(* Logix 5000 project; controller DC01 vendor 1 type 14 code 165 rev 32.12; software revision 32.04; part 8 of 13 *)
(* tags used below, declared in another part *)
   Break1_Length : DINT;
   Break2_Length : DINT;
   Lunch_Length : DINT;
   null : STRING;
   LN03_Schedule : UDT_Current_Status;
   LN03_Weekly_Schedule : UDT_Weekly_Schedule;
(* LN03, continued *)

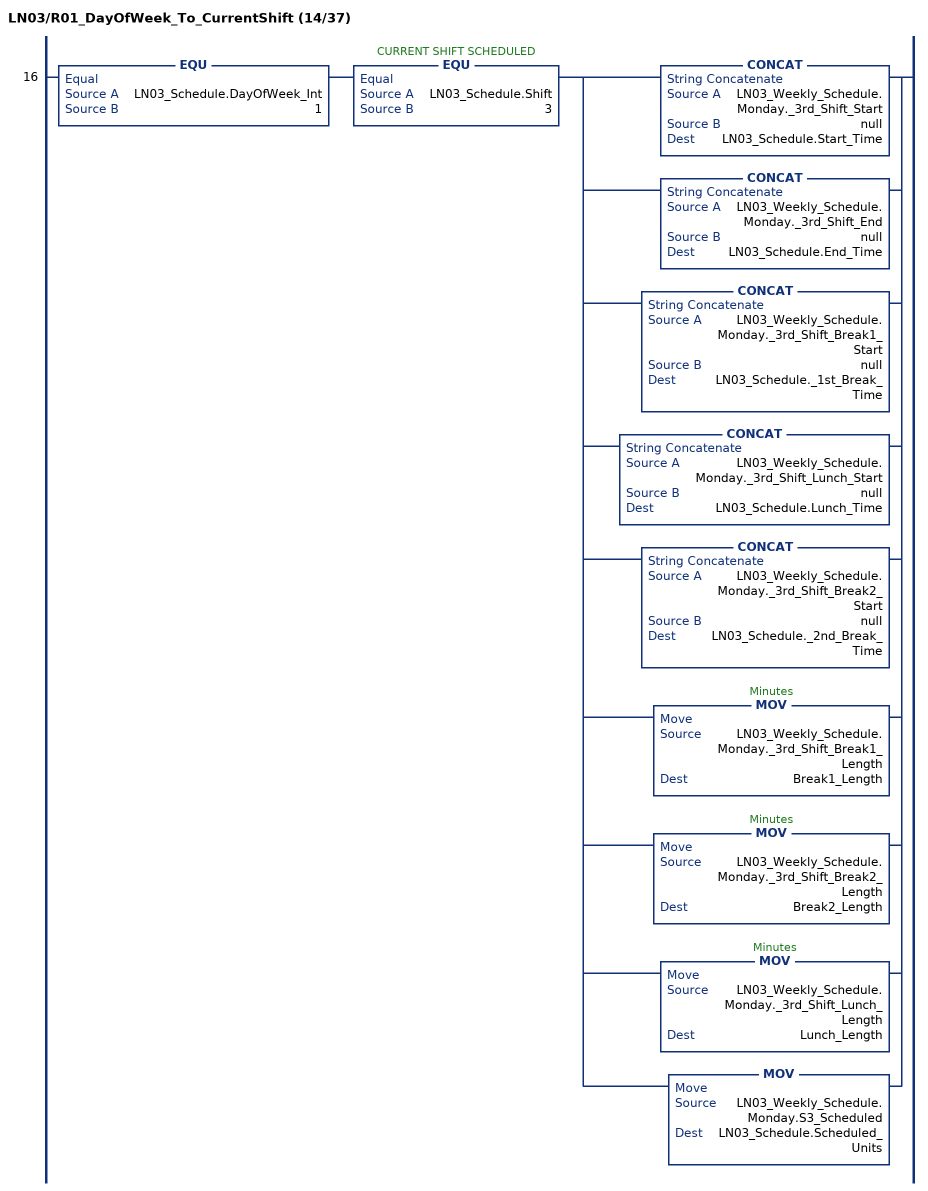
   [picture p147: LN03/R01_DayOfWeek_To_CurrentShift rungs 16-16]
   16: EQU(LN03_Schedule.DayOfWeek_Int,1)EQU(LN03_Schedule.Shift,3)[CONCAT(LN03_Weekly_Schedule.Monday._3rd_Shift_Start,null,LN03_Schedule.Start_Time) ,CONCAT(LN03_Weekly_Schedule.Monday._3rd_Shift_End,null,LN03_Schedule.End_Time) ,CONCAT(LN03_Weekly_Schedule.Monday._3rd_Shift_Break1_Start,null,LN03_Schedule._1st_Break_Time) ,CONCAT(LN03_Weekly_Schedule.Monday._3rd_Shift_Lunch_Start,null,LN03_Schedule.Lunch_Time) ,CONCAT(LN03_Weekly_Schedule.Monday._3rd_Shift_Break2_Start,null,LN03_Schedule._2nd_Break_Time) ,MOV(LN03_Weekly_Schedule.Monday._3rd_Shift_Break1_Length,Break1_Length) ,MOV(LN03_Weekly_Schedule.Monday._3rd_Shift_Break2_Length,Break2_Length) ,MOV(LN03_Weekly_Schedule.Monday._3rd_Shift_Lunch_Length,Lunch_Length) ,MOV(LN03_Weekly_Schedule.Monday.S3_Scheduled,LN03_Schedule.Scheduled_Units) ];
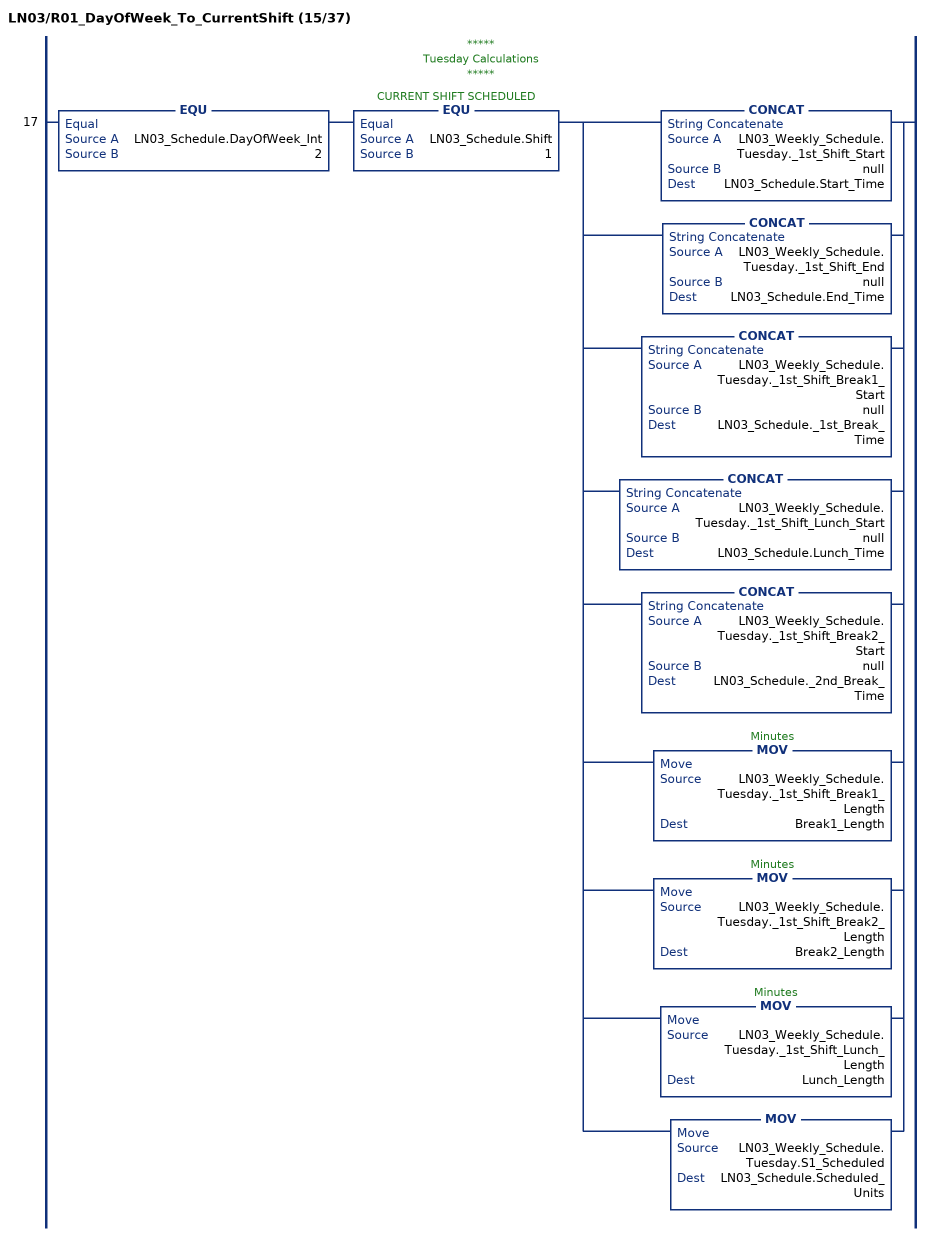
   // *****
   // Tuesday Calculations
   // *****
   17: EQU(LN03_Schedule.DayOfWeek_Int,2)EQU(LN03_Schedule.Shift,1)[CONCAT(LN03_Weekly_Schedule.Tuesday._1st_Shift_Start,null,LN03_Schedule.Start_Time) ,CONCAT(LN03_Weekly_Schedule.Tuesday._1st_Shift_End,null,LN03_Schedule.End_Time) ,CONCAT(LN03_Weekly_Schedule.Tuesday._1st_Shift_Break1_Start,null,LN03_Schedule._1st_Break_Time) ,CONCAT(LN03_Weekly_Schedule.Tuesday._1st_Shift_Lunch_Start,null,LN03_Schedule.Lunch_Time) ,CONCAT(LN03_Weekly_Schedule.Tuesday._1st_Shift_Break2_Start,null,LN03_Schedule._2nd_Break_Time) ,MOV(LN03_Weekly_Schedule.Tuesday._1st_Shift_Break1_Length,Break1_Length) ,MOV(LN03_Weekly_Schedule.Tuesday._1st_Shift_Break2_Length,Break2_Length) ,MOV(LN03_Weekly_Schedule.Tuesday._1st_Shift_Lunch_Length,Lunch_Length) ,MOV(LN03_Weekly_Schedule.Tuesday.S1_Scheduled,LN03_Schedule.Scheduled_Units) ];
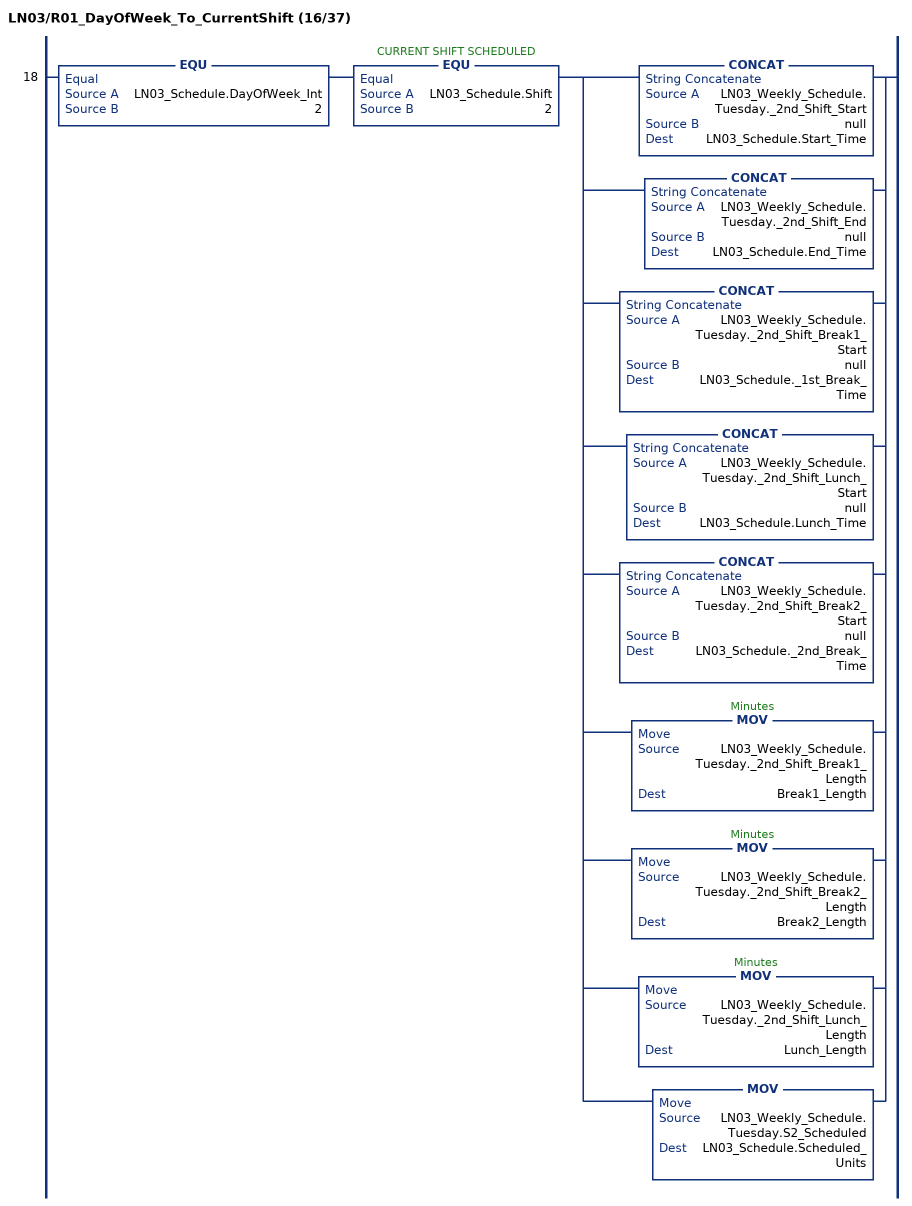
   18: EQU(LN03_Schedule.DayOfWeek_Int,2)EQU(LN03_Schedule.Shift,2)[CONCAT(LN03_Weekly_Schedule.Tuesday._2nd_Shift_Start,null,LN03_Schedule.Start_Time) ,CONCAT(LN03_Weekly_Schedule.Tuesday._2nd_Shift_End,null,LN03_Schedule.End_Time) ,CONCAT(LN03_Weekly_Schedule.Tuesday._2nd_Shift_Break1_Start,null,LN03_Schedule._1st_Break_Time) ,CONCAT(LN03_Weekly_Schedule.Tuesday._2nd_Shift_Lunch_Start,null,LN03_Schedule.Lunch_Time) ,CONCAT(LN03_Weekly_Schedule.Tuesday._2nd_Shift_Break2_Start,null,LN03_Schedule._2nd_Break_Time) ,MOV(LN03_Weekly_Schedule.Tuesday._2nd_Shift_Break1_Length,Break1_Length) ,MOV(LN03_Weekly_Schedule.Tuesday._2nd_Shift_Break2_Length,Break2_Length) ,MOV(LN03_Weekly_Schedule.Tuesday._2nd_Shift_Lunch_Length,Lunch_Length) ,MOV(LN03_Weekly_Schedule.Tuesday.S2_Scheduled,LN03_Schedule.Scheduled_Units) ];
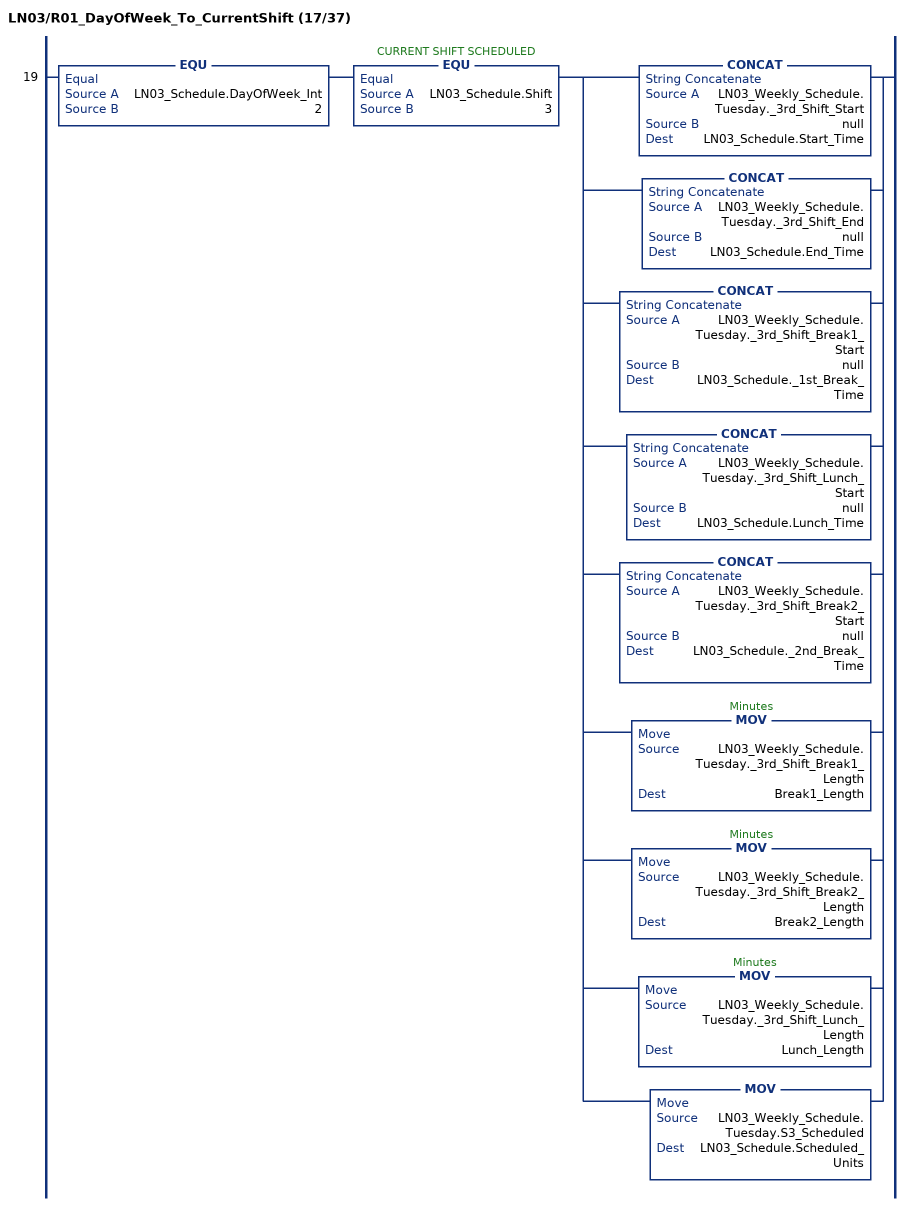
   19: EQU(LN03_Schedule.DayOfWeek_Int,2)EQU(LN03_Schedule.Shift,3)[CONCAT(LN03_Weekly_Schedule.Tuesday._3rd_Shift_Start,null,LN03_Schedule.Start_Time) ,CONCAT(LN03_Weekly_Schedule.Tuesday._3rd_Shift_End,null,LN03_Schedule.End_Time) ,CONCAT(LN03_Weekly_Schedule.Tuesday._3rd_Shift_Break1_Start,null,LN03_Schedule._1st_Break_Time) ,CONCAT(LN03_Weekly_Schedule.Tuesday._3rd_Shift_Lunch_Start,null,LN03_Schedule.Lunch_Time) ,CONCAT(LN03_Weekly_Schedule.Tuesday._3rd_Shift_Break2_Start,null,LN03_Schedule._2nd_Break_Time) ,MOV(LN03_Weekly_Schedule.Tuesday._3rd_Shift_Break1_Length,Break1_Length) ,MOV(LN03_Weekly_Schedule.Tuesday._3rd_Shift_Break2_Length,Break2_Length) ,MOV(LN03_Weekly_Schedule.Tuesday._3rd_Shift_Lunch_Length,Lunch_Length) ,MOV(LN03_Weekly_Schedule.Tuesday.S3_Scheduled,LN03_Schedule.Scheduled_Units) ];
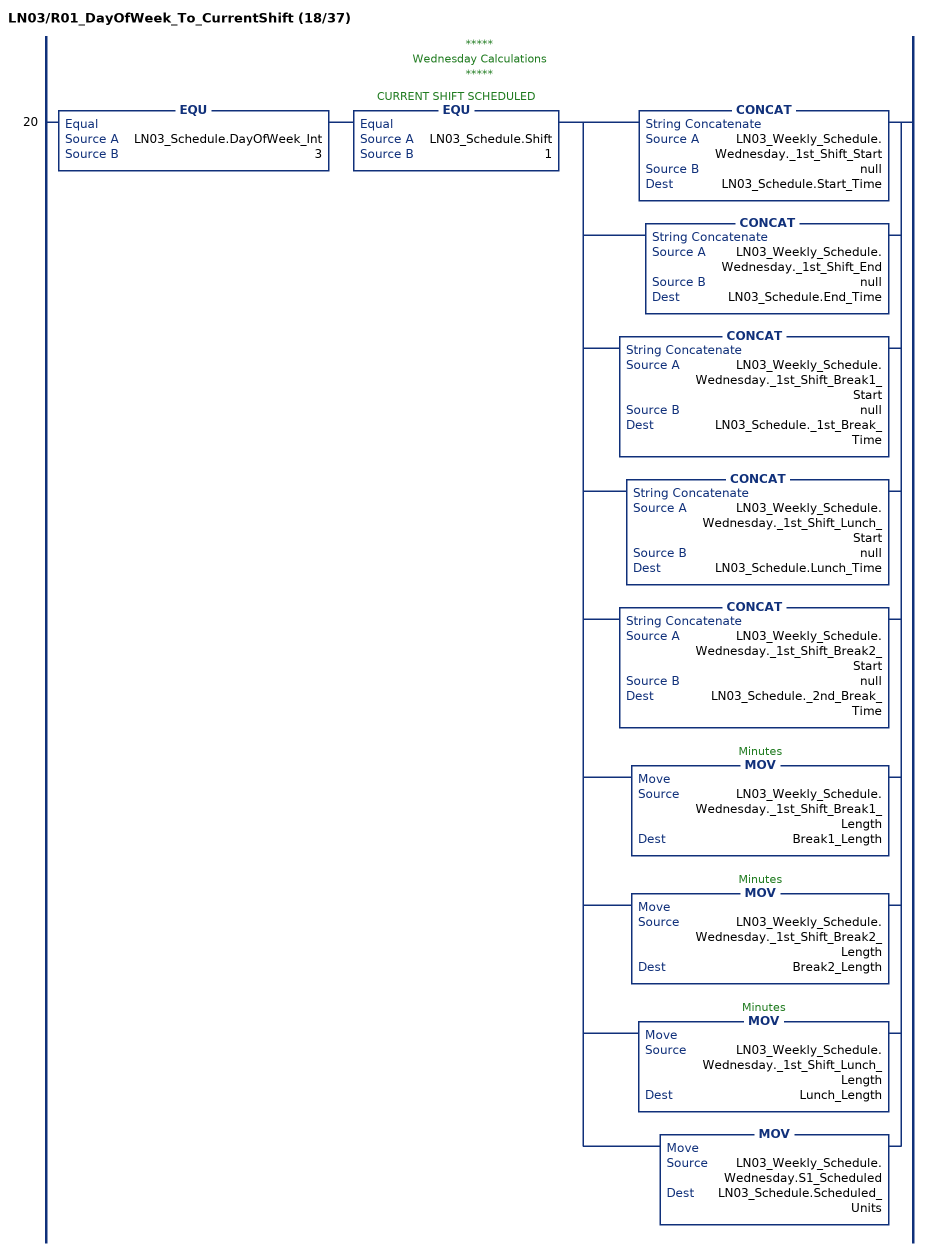
   // *****
   // Wednesday Calculations
   // *****
   20: EQU(LN03_Schedule.DayOfWeek_Int,3)EQU(LN03_Schedule.Shift,1)[CONCAT(LN03_Weekly_Schedule.Wednesday._1st_Shift_Start,null,LN03_Schedule.Start_Time) ,CONCAT(LN03_Weekly_Schedule.Wednesday._1st_Shift_End,null,LN03_Schedule.End_Time) ,CONCAT(LN03_Weekly_Schedule.Wednesday._1st_Shift_Break1_Start,null,LN03_Schedule._1st_Break_Time) ,CONCAT(LN03_Weekly_Schedule.Wednesday._1st_Shift_Lunch_Start,null,LN03_Schedule.Lunch_Time) ,CONCAT(LN03_Weekly_Schedule.Wednesday._1st_Shift_Break2_Start,null,LN03_Schedule._2nd_Break_Time) ,MOV(LN03_Weekly_Schedule.Wednesday._1st_Shift_Break1_Length,Break1_Length) ,MOV(LN03_Weekly_Schedule.Wednesday._1st_Shift_Break2_Length,Break2_Length) ,MOV(LN03_Weekly_Schedule.Wednesday._1st_Shift_Lunch_Length,Lunch_Length) ,MOV(LN03_Weekly_Schedule.Wednesday.S1_Scheduled,LN03_Schedule.Scheduled_Units) ];
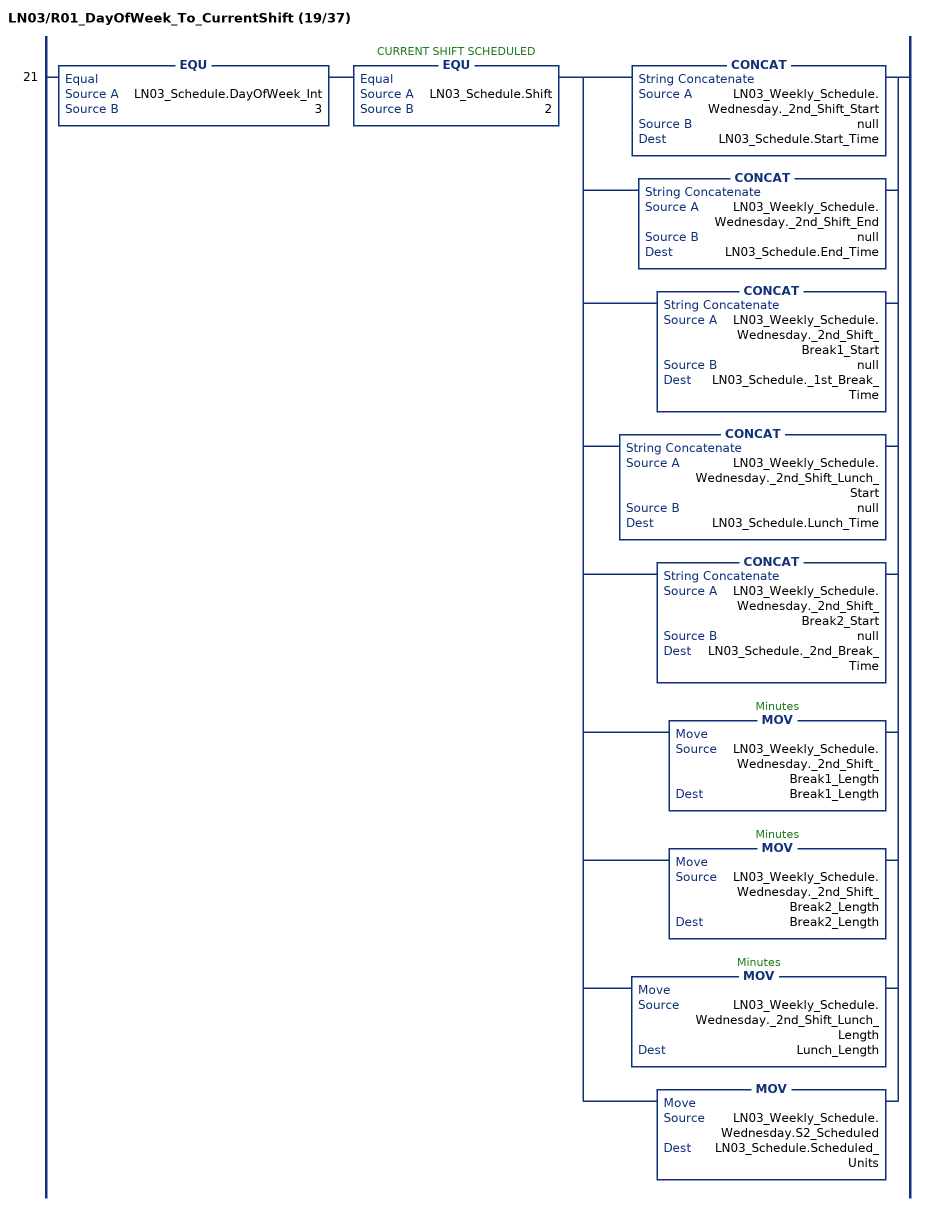
   21: EQU(LN03_Schedule.DayOfWeek_Int,3)EQU(LN03_Schedule.Shift,2)[CONCAT(LN03_Weekly_Schedule.Wednesday._2nd_Shift_Start,null,LN03_Schedule.Start_Time) ,CONCAT(LN03_Weekly_Schedule.Wednesday._2nd_Shift_End,null,LN03_Schedule.End_Time) ,CONCAT(LN03_Weekly_Schedule.Wednesday._2nd_Shift_Break1_Start,null,LN03_Schedule._1st_Break_Time) ,CONCAT(LN03_Weekly_Schedule.Wednesday._2nd_Shift_Lunch_Start,null,LN03_Schedule.Lunch_Time) ,CONCAT(LN03_Weekly_Schedule.Wednesday._2nd_Shift_Break2_Start,null,LN03_Schedule._2nd_Break_Time) ,MOV(LN03_Weekly_Schedule.Wednesday._2nd_Shift_Break1_Length,Break1_Length) ,MOV(LN03_Weekly_Schedule.Wednesday._2nd_Shift_Break2_Length,Break2_Length) ,MOV(LN03_Weekly_Schedule.Wednesday._2nd_Shift_Lunch_Length,Lunch_Length) ,MOV(LN03_Weekly_Schedule.Wednesday.S2_Scheduled,LN03_Schedule.Scheduled_Units) ];
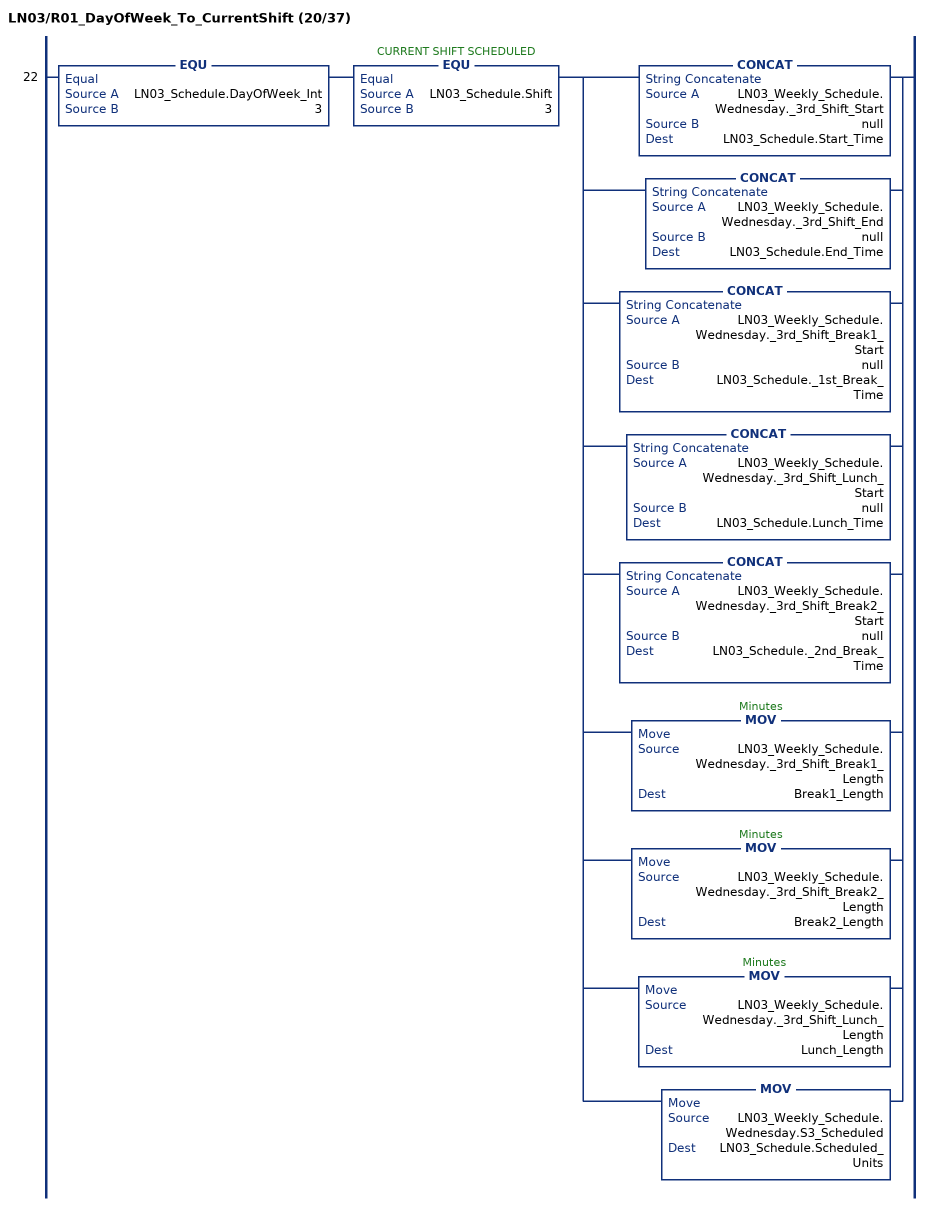
   22: EQU(LN03_Schedule.DayOfWeek_Int,3)EQU(LN03_Schedule.Shift,3)[CONCAT(LN03_Weekly_Schedule.Wednesday._3rd_Shift_Start,null,LN03_Schedule.Start_Time) ,CONCAT(LN03_Weekly_Schedule.Wednesday._3rd_Shift_End,null,LN03_Schedule.End_Time) ,CONCAT(LN03_Weekly_Schedule.Wednesday._3rd_Shift_Break1_Start,null,LN03_Schedule._1st_Break_Time) ,CONCAT(LN03_Weekly_Schedule.Wednesday._3rd_Shift_Lunch_Start,null,LN03_Schedule.Lunch_Time) ,CONCAT(LN03_Weekly_Schedule.Wednesday._3rd_Shift_Break2_Start,null,LN03_Schedule._2nd_Break_Time) ,MOV(LN03_Weekly_Schedule.Wednesday._3rd_Shift_Break1_Length,Break1_Length) ,MOV(LN03_Weekly_Schedule.Wednesday._3rd_Shift_Break2_Length,Break2_Length) ,MOV(LN03_Weekly_Schedule.Wednesday._3rd_Shift_Lunch_Length,Lunch_Length) ,MOV(LN03_Weekly_Schedule.Wednesday.S3_Scheduled,LN03_Schedule.Scheduled_Units) ];
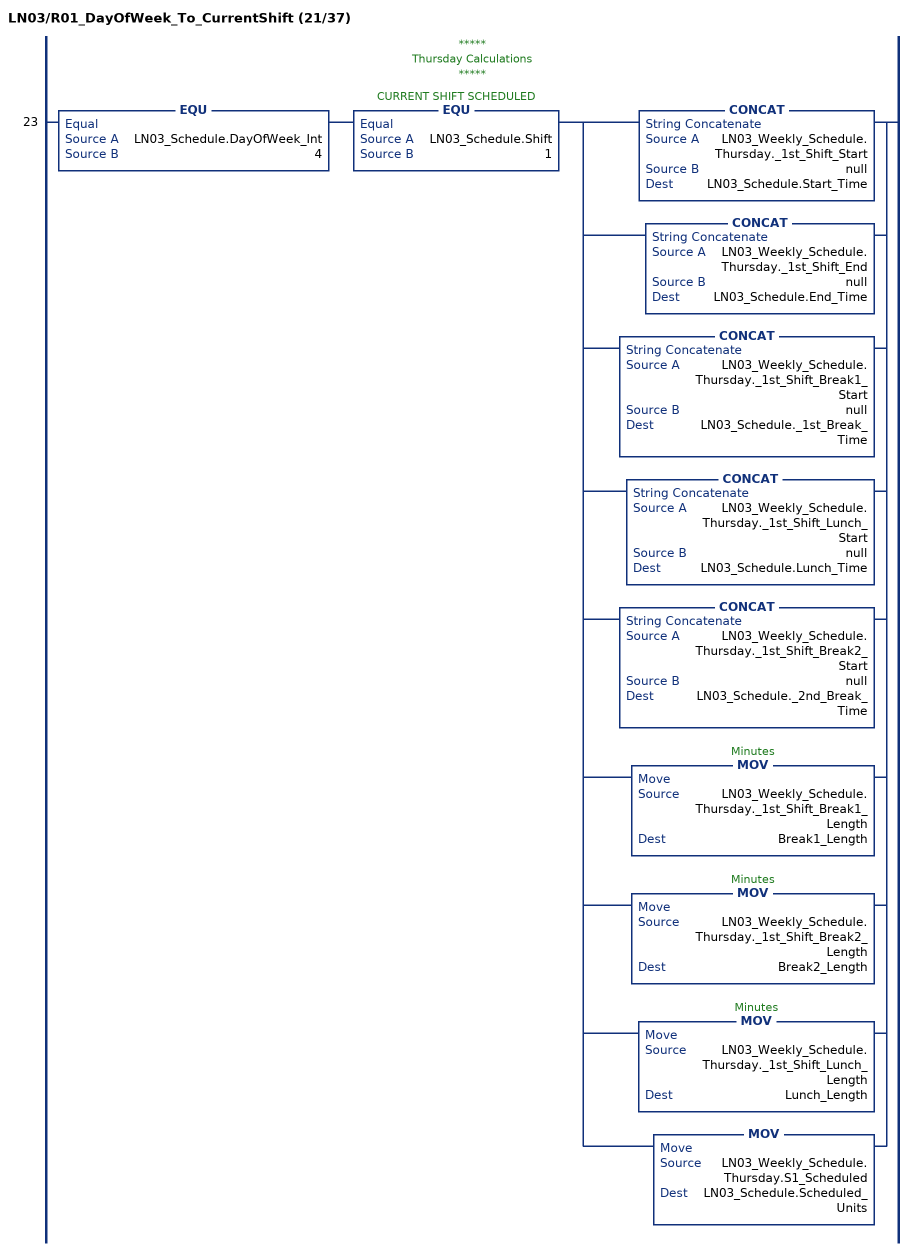
   // *****
   // Thursday Calculations
   // *****
   23: EQU(LN03_Schedule.DayOfWeek_Int,4)EQU(LN03_Schedule.Shift,1)[CONCAT(LN03_Weekly_Schedule.Thursday._1st_Shift_Start,null,LN03_Schedule.Start_Time) ,CONCAT(LN03_Weekly_Schedule.Thursday._1st_Shift_End,null,LN03_Schedule.End_Time) ,CONCAT(LN03_Weekly_Schedule.Thursday._1st_Shift_Break1_Start,null,LN03_Schedule._1st_Break_Time) ,CONCAT(LN03_Weekly_Schedule.Thursday._1st_Shift_Lunch_Start,null,LN03_Schedule.Lunch_Time) ,CONCAT(LN03_Weekly_Schedule.Thursday._1st_Shift_Break2_Start,null,LN03_Schedule._2nd_Break_Time) ,MOV(LN03_Weekly_Schedule.Thursday._1st_Shift_Break1_Length,Break1_Length) ,MOV(LN03_Weekly_Schedule.Thursday._1st_Shift_Break2_Length,Break2_Length) ,MOV(LN03_Weekly_Schedule.Thursday._1st_Shift_Lunch_Length,Lunch_Length) ,MOV(LN03_Weekly_Schedule.Thursday.S1_Scheduled,LN03_Schedule.Scheduled_Units) ];
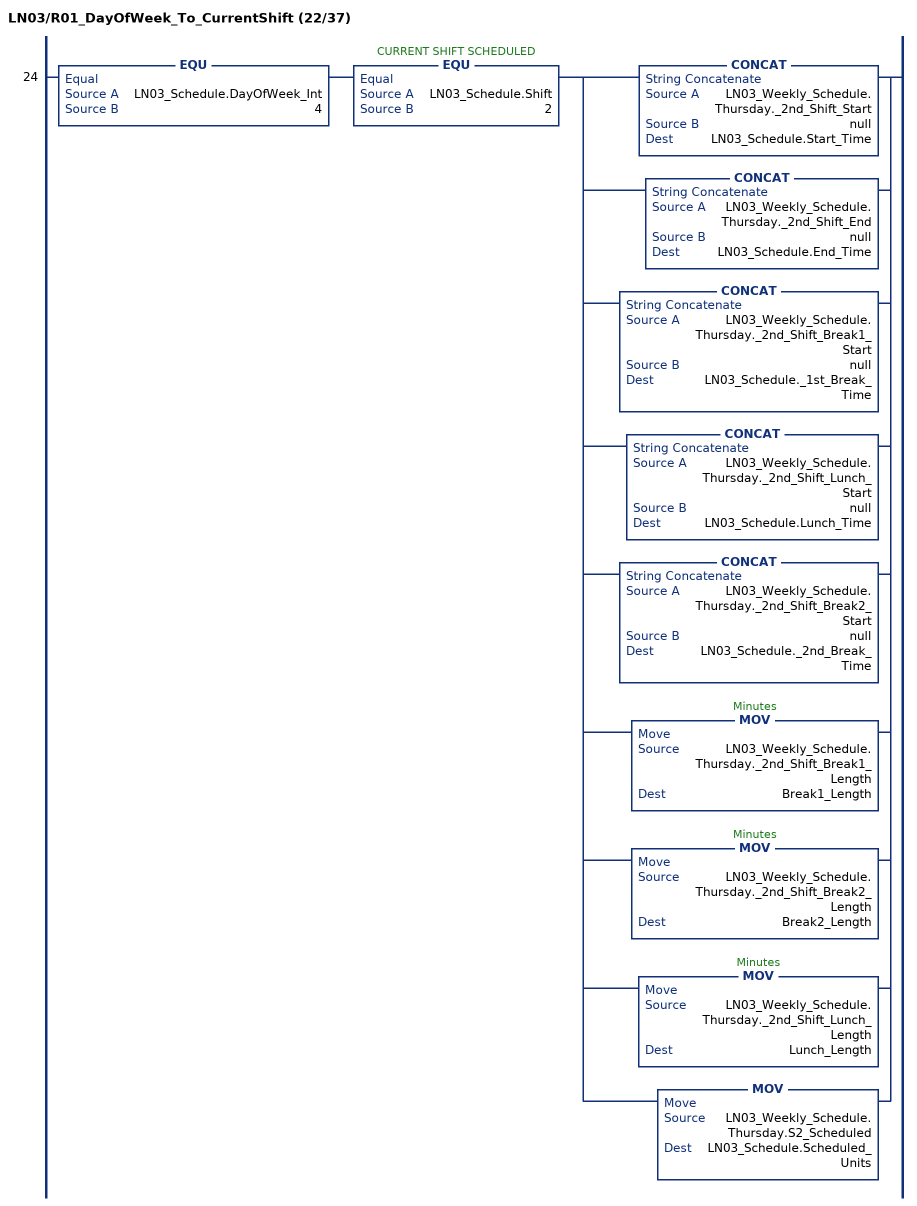
   24: EQU(LN03_Schedule.DayOfWeek_Int,4)EQU(LN03_Schedule.Shift,2)[CONCAT(LN03_Weekly_Schedule.Thursday._2nd_Shift_Start,null,LN03_Schedule.Start_Time) ,CONCAT(LN03_Weekly_Schedule.Thursday._2nd_Shift_End,null,LN03_Schedule.End_Time) ,CONCAT(LN03_Weekly_Schedule.Thursday._2nd_Shift_Break1_Start,null,LN03_Schedule._1st_Break_Time) ,CONCAT(LN03_Weekly_Schedule.Thursday._2nd_Shift_Lunch_Start,null,LN03_Schedule.Lunch_Time) ,CONCAT(LN03_Weekly_Schedule.Thursday._2nd_Shift_Break2_Start,null,LN03_Schedule._2nd_Break_Time) ,MOV(LN03_Weekly_Schedule.Thursday._2nd_Shift_Break1_Length,Break1_Length) ,MOV(LN03_Weekly_Schedule.Thursday._2nd_Shift_Break2_Length,Break2_Length) ,MOV(LN03_Weekly_Schedule.Thursday._2nd_Shift_Lunch_Length,Lunch_Length) ,MOV(LN03_Weekly_Schedule.Thursday.S2_Scheduled,LN03_Schedule.Scheduled_Units) ];
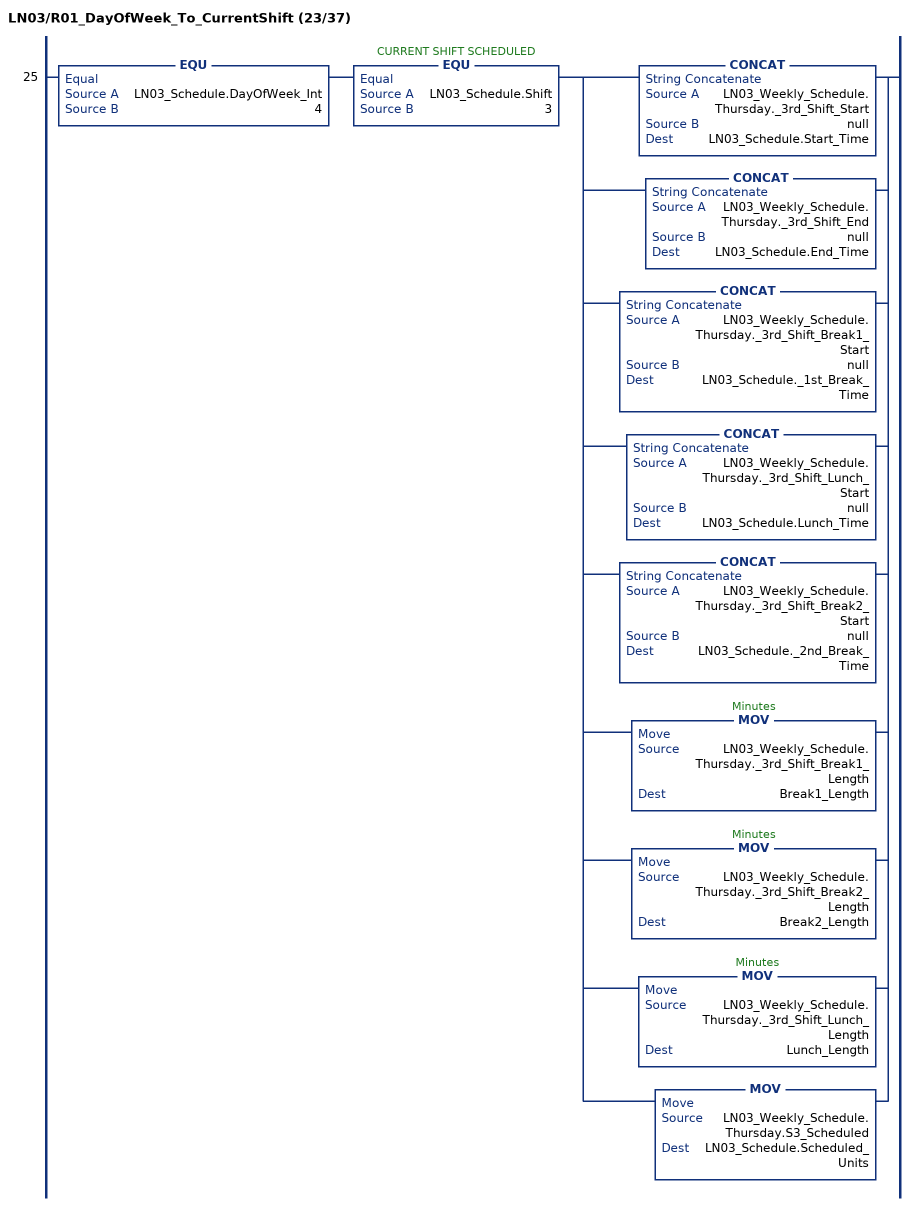
   25: EQU(LN03_Schedule.DayOfWeek_Int,4)EQU(LN03_Schedule.Shift,3)[CONCAT(LN03_Weekly_Schedule.Thursday._3rd_Shift_Start,null,LN03_Schedule.Start_Time) ,CONCAT(LN03_Weekly_Schedule.Thursday._3rd_Shift_End,null,LN03_Schedule.End_Time) ,CONCAT(LN03_Weekly_Schedule.Thursday._3rd_Shift_Break1_Start,null,LN03_Schedule._1st_Break_Time) ,CONCAT(LN03_Weekly_Schedule.Thursday._3rd_Shift_Lunch_Start,null,LN03_Schedule.Lunch_Time) ,CONCAT(LN03_Weekly_Schedule.Thursday._3rd_Shift_Break2_Start,null,LN03_Schedule._2nd_Break_Time) ,MOV(LN03_Weekly_Schedule.Thursday._3rd_Shift_Break1_Length,Break1_Length) ,MOV(LN03_Weekly_Schedule.Thursday._3rd_Shift_Break2_Length,Break2_Length) ,MOV(LN03_Weekly_Schedule.Thursday._3rd_Shift_Lunch_Length,Lunch_Length) ,MOV(LN03_Weekly_Schedule.Thursday.S3_Scheduled,LN03_Schedule.Scheduled_Units) ];
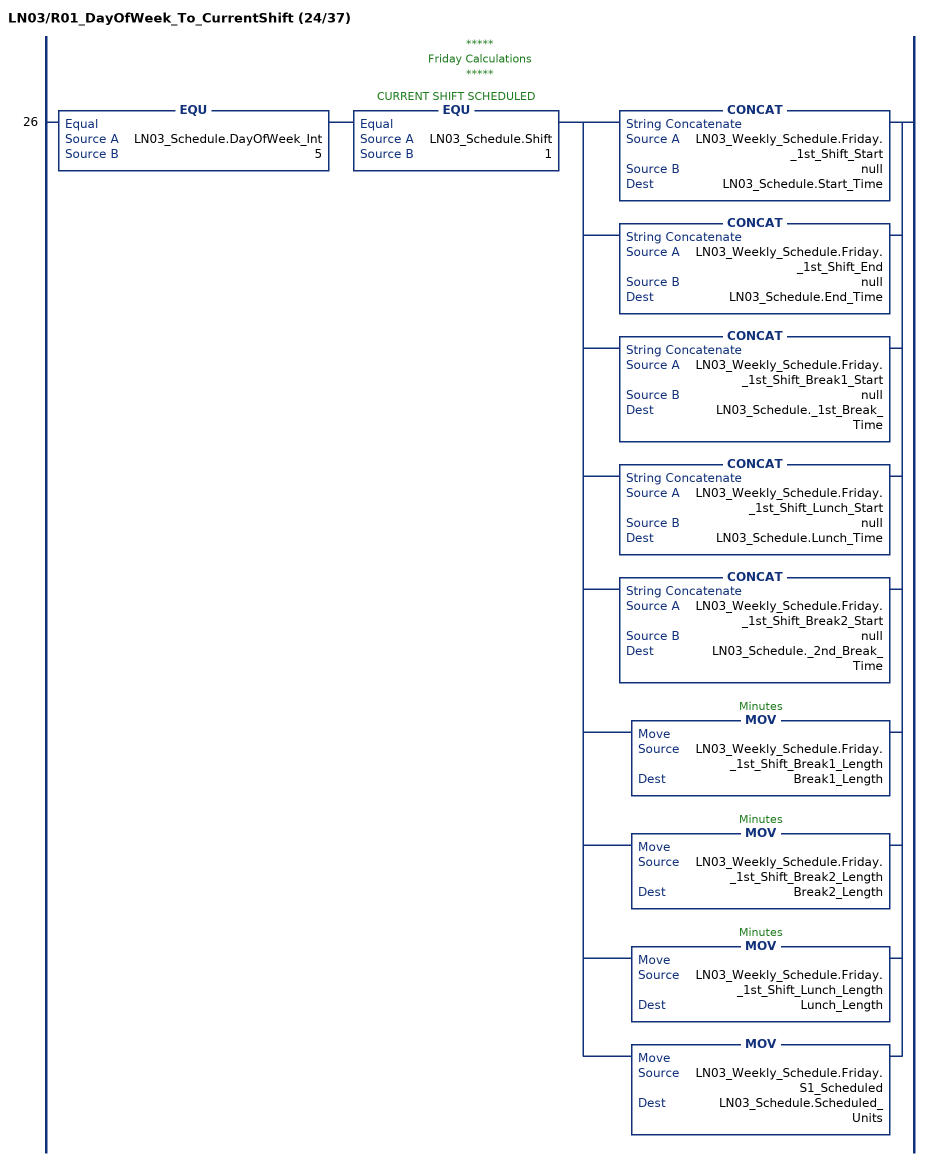
   // *****
   // Friday Calculations
   // *****
   26: EQU(LN03_Schedule.DayOfWeek_Int,5)EQU(LN03_Schedule.Shift,1)[CONCAT(LN03_Weekly_Schedule.Friday._1st_Shift_Start,null,LN03_Schedule.Start_Time) ,CONCAT(LN03_Weekly_Schedule.Friday._1st_Shift_End,null,LN03_Schedule.End_Time) ,CONCAT(LN03_Weekly_Schedule.Friday._1st_Shift_Break1_Start,null,LN03_Schedule._1st_Break_Time) ,CONCAT(LN03_Weekly_Schedule.Friday._1st_Shift_Lunch_Start,null,LN03_Schedule.Lunch_Time) ,CONCAT(LN03_Weekly_Schedule.Friday._1st_Shift_Break2_Start,null,LN03_Schedule._2nd_Break_Time) ,MOV(LN03_Weekly_Schedule.Friday._1st_Shift_Break1_Length,Break1_Length) ,MOV(LN03_Weekly_Schedule.Friday._1st_Shift_Break2_Length,Break2_Length) ,MOV(LN03_Weekly_Schedule.Friday._1st_Shift_Lunch_Length,Lunch_Length) ,MOV(LN03_Weekly_Schedule.Friday.S1_Scheduled,LN03_Schedule.Scheduled_Units) ];
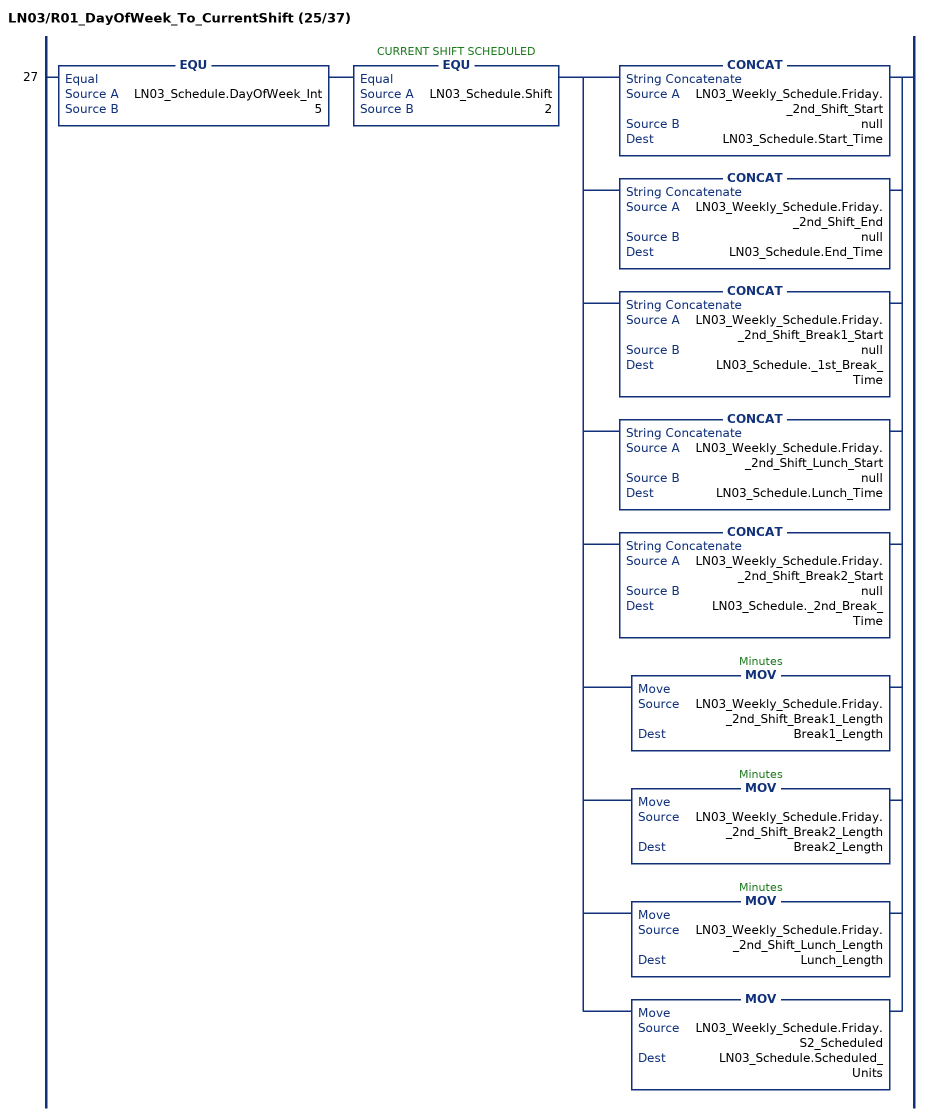
   27: EQU(LN03_Schedule.DayOfWeek_Int,5)EQU(LN03_Schedule.Shift,2)[CONCAT(LN03_Weekly_Schedule.Friday._2nd_Shift_Start,null,LN03_Schedule.Start_Time) ,CONCAT(LN03_Weekly_Schedule.Friday._2nd_Shift_End,null,LN03_Schedule.End_Time) ,CONCAT(LN03_Weekly_Schedule.Friday._2nd_Shift_Break1_Start,null,LN03_Schedule._1st_Break_Time) ,CONCAT(LN03_Weekly_Schedule.Friday._2nd_Shift_Lunch_Start,null,LN03_Schedule.Lunch_Time) ,CONCAT(LN03_Weekly_Schedule.Friday._2nd_Shift_Break2_Start,null,LN03_Schedule._2nd_Break_Time) ,MOV(LN03_Weekly_Schedule.Friday._2nd_Shift_Break1_Length,Break1_Length) ,MOV(LN03_Weekly_Schedule.Friday._2nd_Shift_Break2_Length,Break2_Length) ,MOV(LN03_Weekly_Schedule.Friday._2nd_Shift_Lunch_Length,Lunch_Length) ,MOV(LN03_Weekly_Schedule.Friday.S2_Scheduled,LN03_Schedule.Scheduled_Units) ];
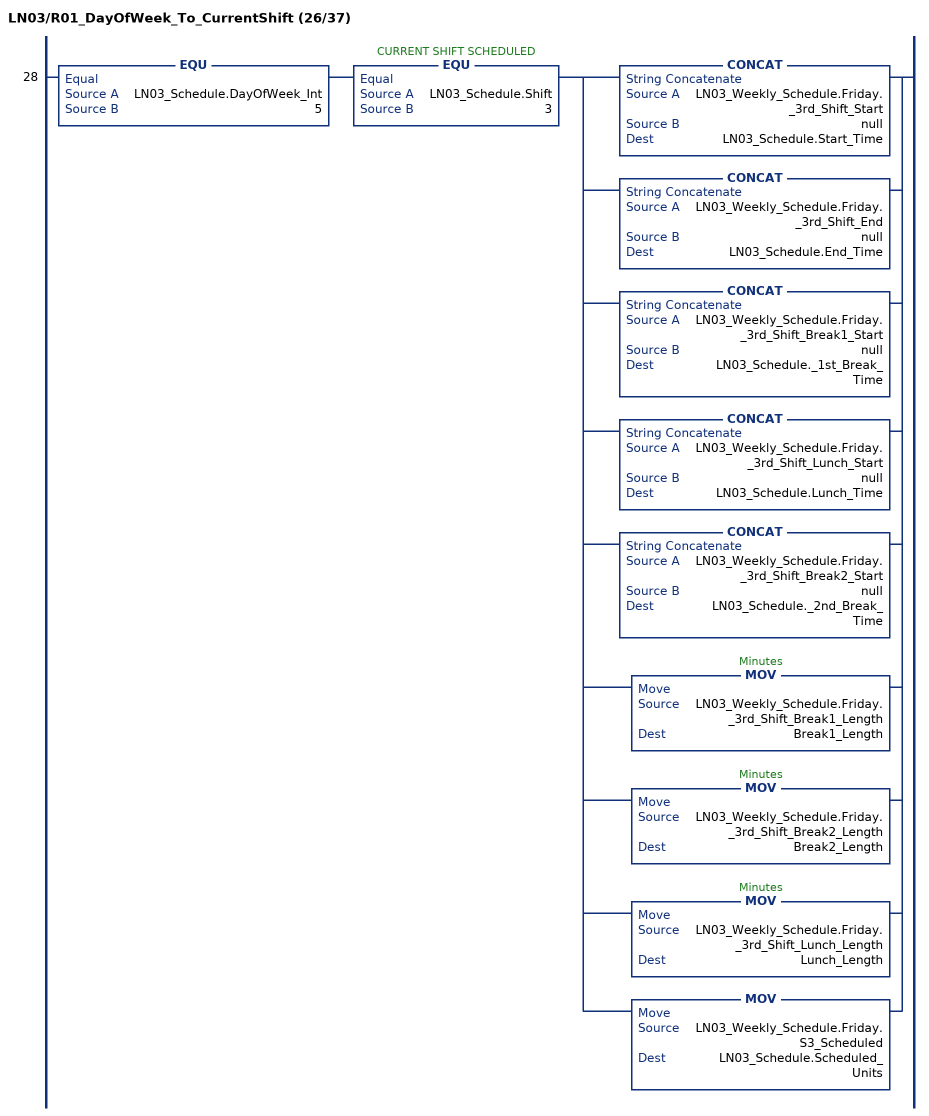
   28: EQU(LN03_Schedule.DayOfWeek_Int,5)EQU(LN03_Schedule.Shift,3)[CONCAT(LN03_Weekly_Schedule.Friday._3rd_Shift_Start,null,LN03_Schedule.Start_Time) ,CONCAT(LN03_Weekly_Schedule.Friday._3rd_Shift_End,null,LN03_Schedule.End_Time) ,CONCAT(LN03_Weekly_Schedule.Friday._3rd_Shift_Break1_Start,null,LN03_Schedule._1st_Break_Time) ,CONCAT(LN03_Weekly_Schedule.Friday._3rd_Shift_Lunch_Start,null,LN03_Schedule.Lunch_Time) ,CONCAT(LN03_Weekly_Schedule.Friday._3rd_Shift_Break2_Start,null,LN03_Schedule._2nd_Break_Time) ,MOV(LN03_Weekly_Schedule.Friday._3rd_Shift_Break1_Length,Break1_Length) ,MOV(LN03_Weekly_Schedule.Friday._3rd_Shift_Break2_Length,Break2_Length) ,MOV(LN03_Weekly_Schedule.Friday._3rd_Shift_Lunch_Length,Lunch_Length) ,MOV(LN03_Weekly_Schedule.Friday.S3_Scheduled,LN03_Schedule.Scheduled_Units) ];
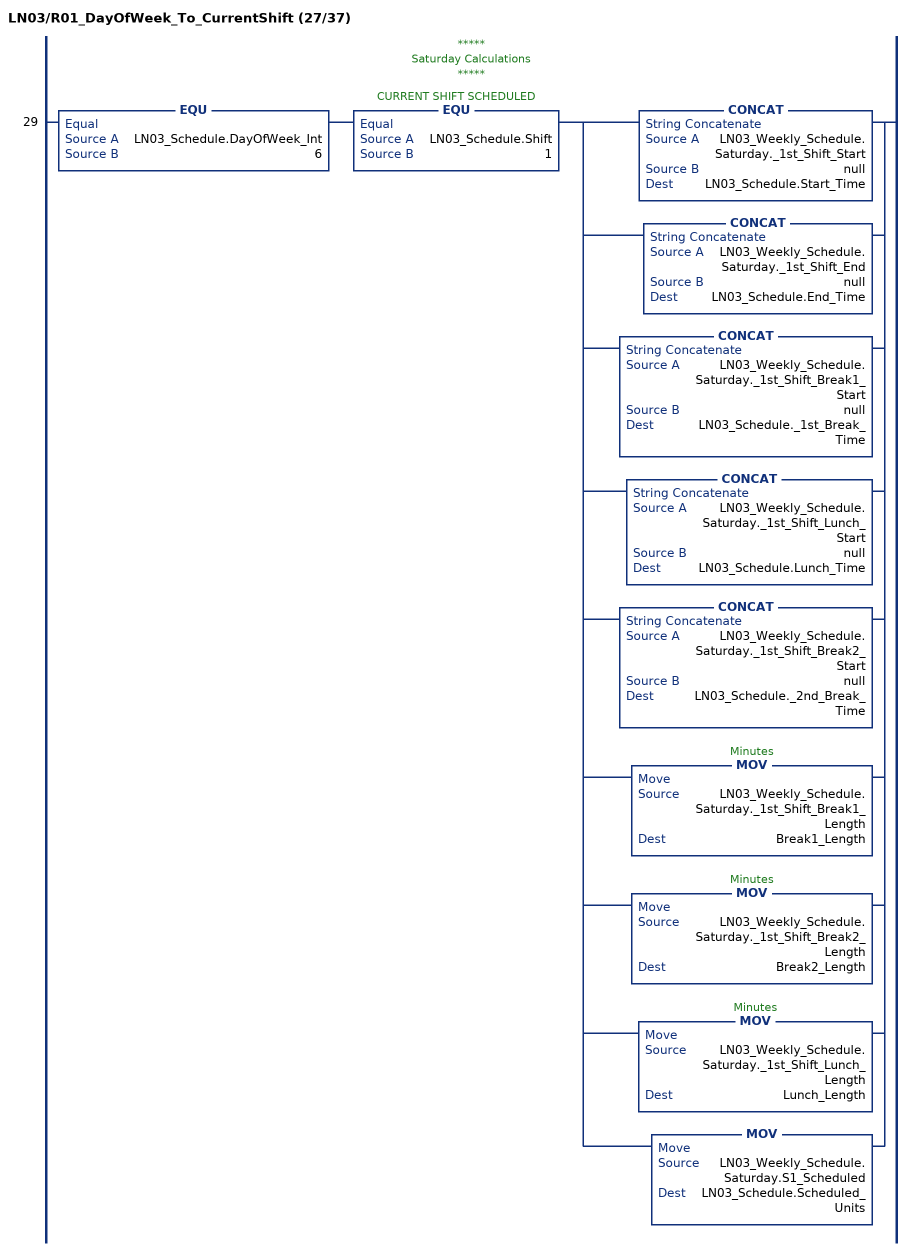
   // *****
   // Saturday Calculations
   // *****
   29: EQU(LN03_Schedule.DayOfWeek_Int,6)EQU(LN03_Schedule.Shift,1)[CONCAT(LN03_Weekly_Schedule.Saturday._1st_Shift_Start,null,LN03_Schedule.Start_Time) ,CONCAT(LN03_Weekly_Schedule.Saturday._1st_Shift_End,null,LN03_Schedule.End_Time) ,CONCAT(LN03_Weekly_Schedule.Saturday._1st_Shift_Break1_Start,null,LN03_Schedule._1st_Break_Time) ,CONCAT(LN03_Weekly_Schedule.Saturday._1st_Shift_Lunch_Start,null,LN03_Schedule.Lunch_Time) ,CONCAT(LN03_Weekly_Schedule.Saturday._1st_Shift_Break2_Start,null,LN03_Schedule._2nd_Break_Time) ,MOV(LN03_Weekly_Schedule.Saturday._1st_Shift_Break1_Length,Break1_Length) ,MOV(LN03_Weekly_Schedule.Saturday._1st_Shift_Break2_Length,Break2_Length) ,MOV(LN03_Weekly_Schedule.Saturday._1st_Shift_Lunch_Length,Lunch_Length) ,MOV(LN03_Weekly_Schedule.Saturday.S1_Scheduled,LN03_Schedule.Scheduled_Units) ];
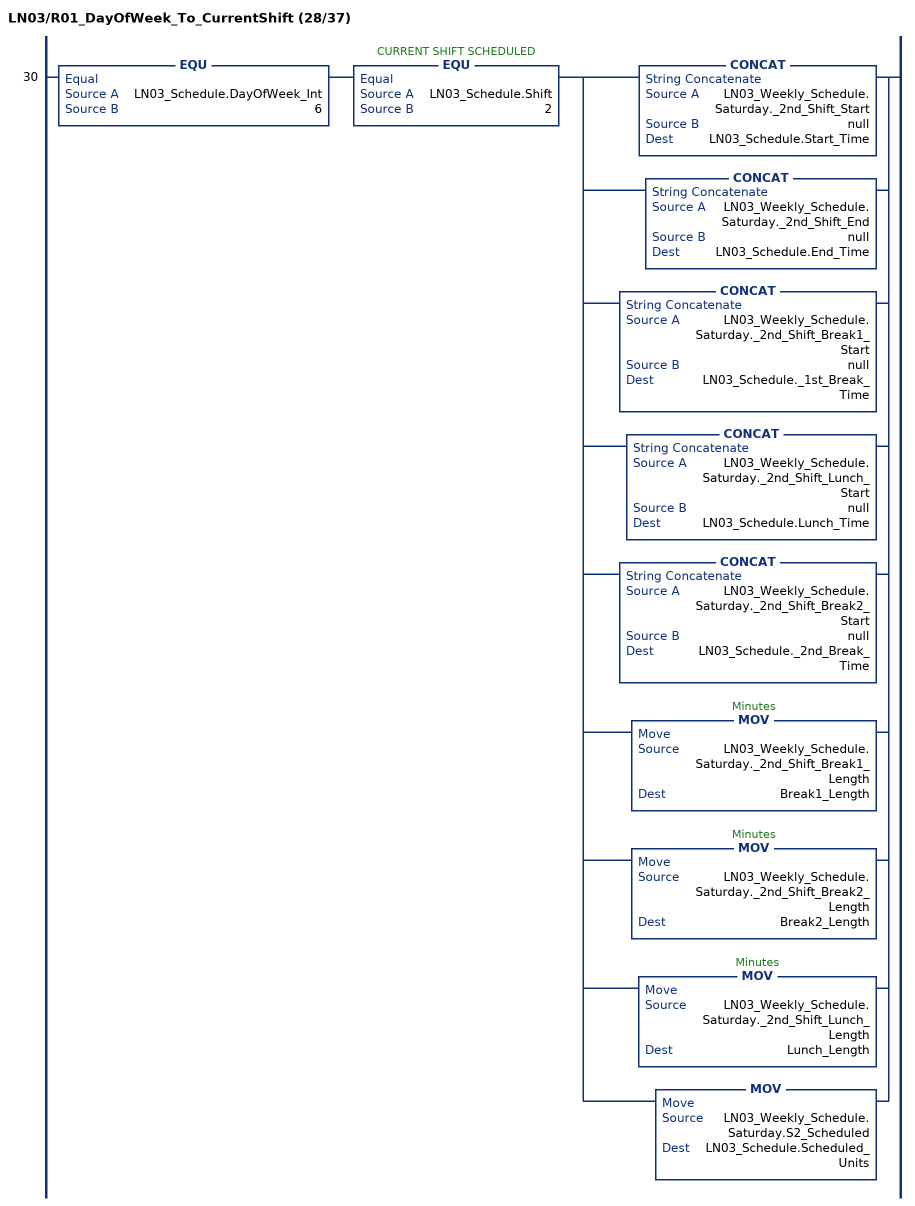
   30: EQU(LN03_Schedule.DayOfWeek_Int,6)EQU(LN03_Schedule.Shift,2)[CONCAT(LN03_Weekly_Schedule.Saturday._2nd_Shift_Start,null,LN03_Schedule.Start_Time) ,CONCAT(LN03_Weekly_Schedule.Saturday._2nd_Shift_End,null,LN03_Schedule.End_Time) ,CONCAT(LN03_Weekly_Schedule.Saturday._2nd_Shift_Break1_Start,null,LN03_Schedule._1st_Break_Time) ,CONCAT(LN03_Weekly_Schedule.Saturday._2nd_Shift_Lunch_Start,null,LN03_Schedule.Lunch_Time) ,CONCAT(LN03_Weekly_Schedule.Saturday._2nd_Shift_Break2_Start,null,LN03_Schedule._2nd_Break_Time) ,MOV(LN03_Weekly_Schedule.Saturday._2nd_Shift_Break1_Length,Break1_Length) ,MOV(LN03_Weekly_Schedule.Saturday._2nd_Shift_Break2_Length,Break2_Length) ,MOV(LN03_Weekly_Schedule.Saturday._2nd_Shift_Lunch_Length,Lunch_Length) ,MOV(LN03_Weekly_Schedule.Saturday.S2_Scheduled,LN03_Schedule.Scheduled_Units) ];
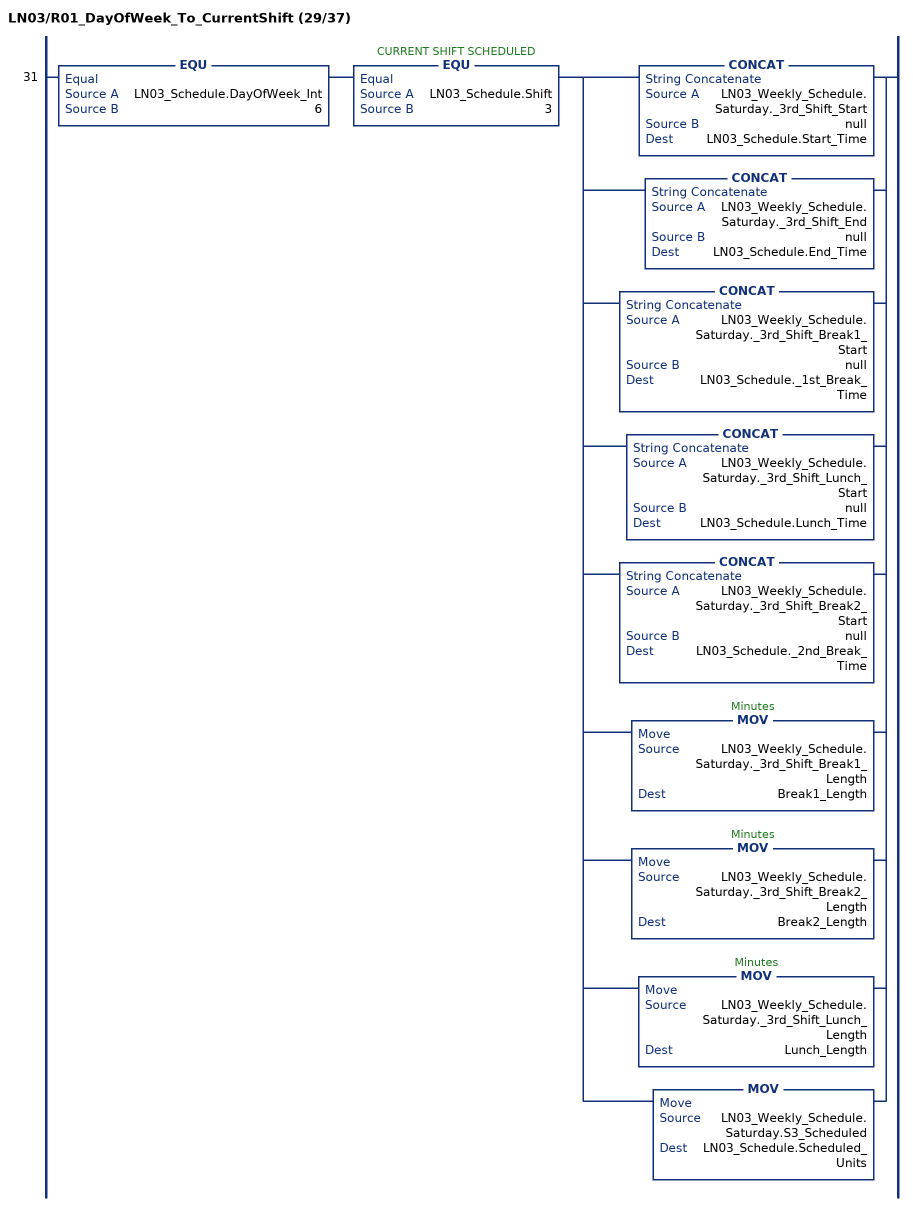
   31: EQU(LN03_Schedule.DayOfWeek_Int,6)EQU(LN03_Schedule.Shift,3)[CONCAT(LN03_Weekly_Schedule.Saturday._3rd_Shift_Start,null,LN03_Schedule.Start_Time) ,CONCAT(LN03_Weekly_Schedule.Saturday._3rd_Shift_End,null,LN03_Schedule.End_Time) ,CONCAT(LN03_Weekly_Schedule.Saturday._3rd_Shift_Break1_Start,null,LN03_Schedule._1st_Break_Time) ,CONCAT(LN03_Weekly_Schedule.Saturday._3rd_Shift_Lunch_Start,null,LN03_Schedule.Lunch_Time) ,CONCAT(LN03_Weekly_Schedule.Saturday._3rd_Shift_Break2_Start,null,LN03_Schedule._2nd_Break_Time) ,MOV(LN03_Weekly_Schedule.Saturday._3rd_Shift_Break1_Length,Break1_Length) ,MOV(LN03_Weekly_Schedule.Saturday._3rd_Shift_Break2_Length,Break2_Length) ,MOV(LN03_Weekly_Schedule.Saturday._3rd_Shift_Lunch_Length,Lunch_Length) ,MOV(LN03_Weekly_Schedule.Saturday.S3_Scheduled,LN03_Schedule.Scheduled_Units) ];
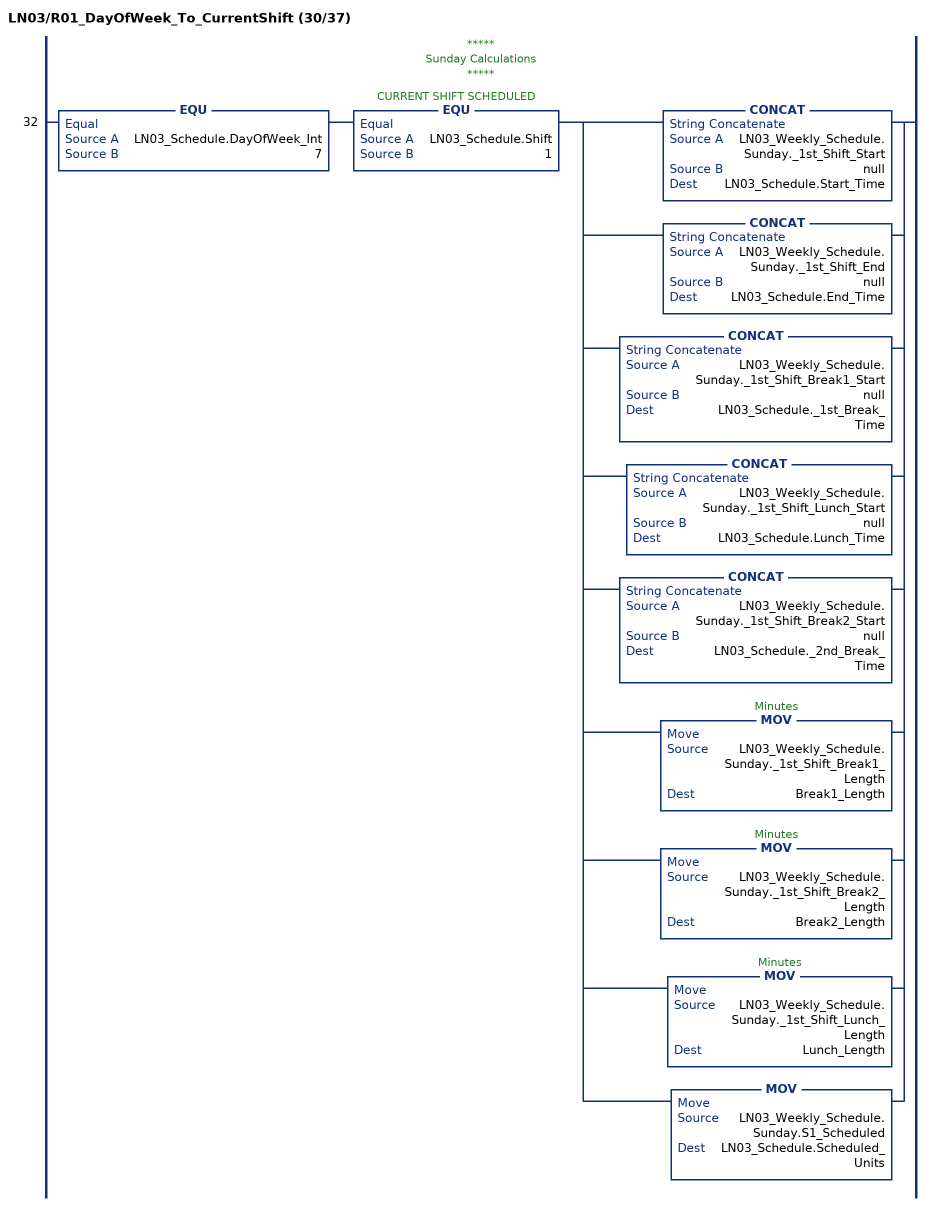
   // *****
   // Sunday Calculations
   // *****
   32: EQU(LN03_Schedule.DayOfWeek_Int,7)EQU(LN03_Schedule.Shift,1)[CONCAT(LN03_Weekly_Schedule.Sunday._1st_Shift_Start,null,LN03_Schedule.Start_Time) ,CONCAT(LN03_Weekly_Schedule.Sunday._1st_Shift_End,null,LN03_Schedule.End_Time) ,CONCAT(LN03_Weekly_Schedule.Sunday._1st_Shift_Break1_Start,null,LN03_Schedule._1st_Break_Time) ,CONCAT(LN03_Weekly_Schedule.Sunday._1st_Shift_Lunch_Start,null,LN03_Schedule.Lunch_Time) ,CONCAT(LN03_Weekly_Schedule.Sunday._1st_Shift_Break2_Start,null,LN03_Schedule._2nd_Break_Time) ,MOV(LN03_Weekly_Schedule.Sunday._1st_Shift_Break1_Length,Break1_Length) ,MOV(LN03_Weekly_Schedule.Sunday._1st_Shift_Break2_Length,Break2_Length) ,MOV(LN03_Weekly_Schedule.Sunday._1st_Shift_Lunch_Length,Lunch_Length) ,MOV(LN03_Weekly_Schedule.Sunday.S1_Scheduled,LN03_Schedule.Scheduled_Units) ];
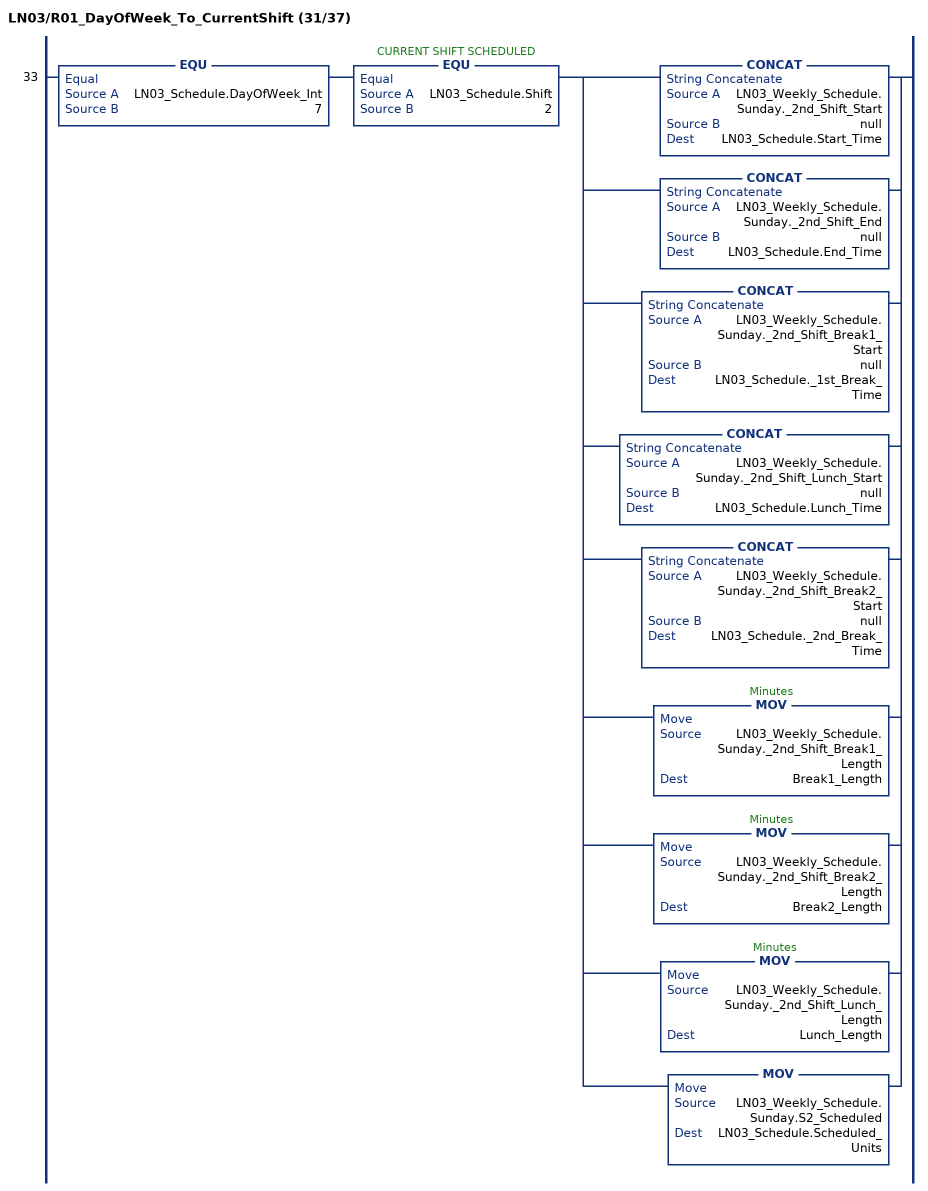
   33: EQU(LN03_Schedule.DayOfWeek_Int,7)EQU(LN03_Schedule.Shift,2)[CONCAT(LN03_Weekly_Schedule.Sunday._2nd_Shift_Start,null,LN03_Schedule.Start_Time) ,CONCAT(LN03_Weekly_Schedule.Sunday._2nd_Shift_End,null,LN03_Schedule.End_Time) ,CONCAT(LN03_Weekly_Schedule.Sunday._2nd_Shift_Break1_Start,null,LN03_Schedule._1st_Break_Time) ,CONCAT(LN03_Weekly_Schedule.Sunday._2nd_Shift_Lunch_Start,null,LN03_Schedule.Lunch_Time) ,CONCAT(LN03_Weekly_Schedule.Sunday._2nd_Shift_Break2_Start,null,LN03_Schedule._2nd_Break_Time) ,MOV(LN03_Weekly_Schedule.Sunday._2nd_Shift_Break1_Length,Break1_Length) ,MOV(LN03_Weekly_Schedule.Sunday._2nd_Shift_Break2_Length,Break2_Length) ,MOV(LN03_Weekly_Schedule.Sunday._2nd_Shift_Lunch_Length,Lunch_Length) ,MOV(LN03_Weekly_Schedule.Sunday.S2_Scheduled,LN03_Schedule.Scheduled_Units) ];
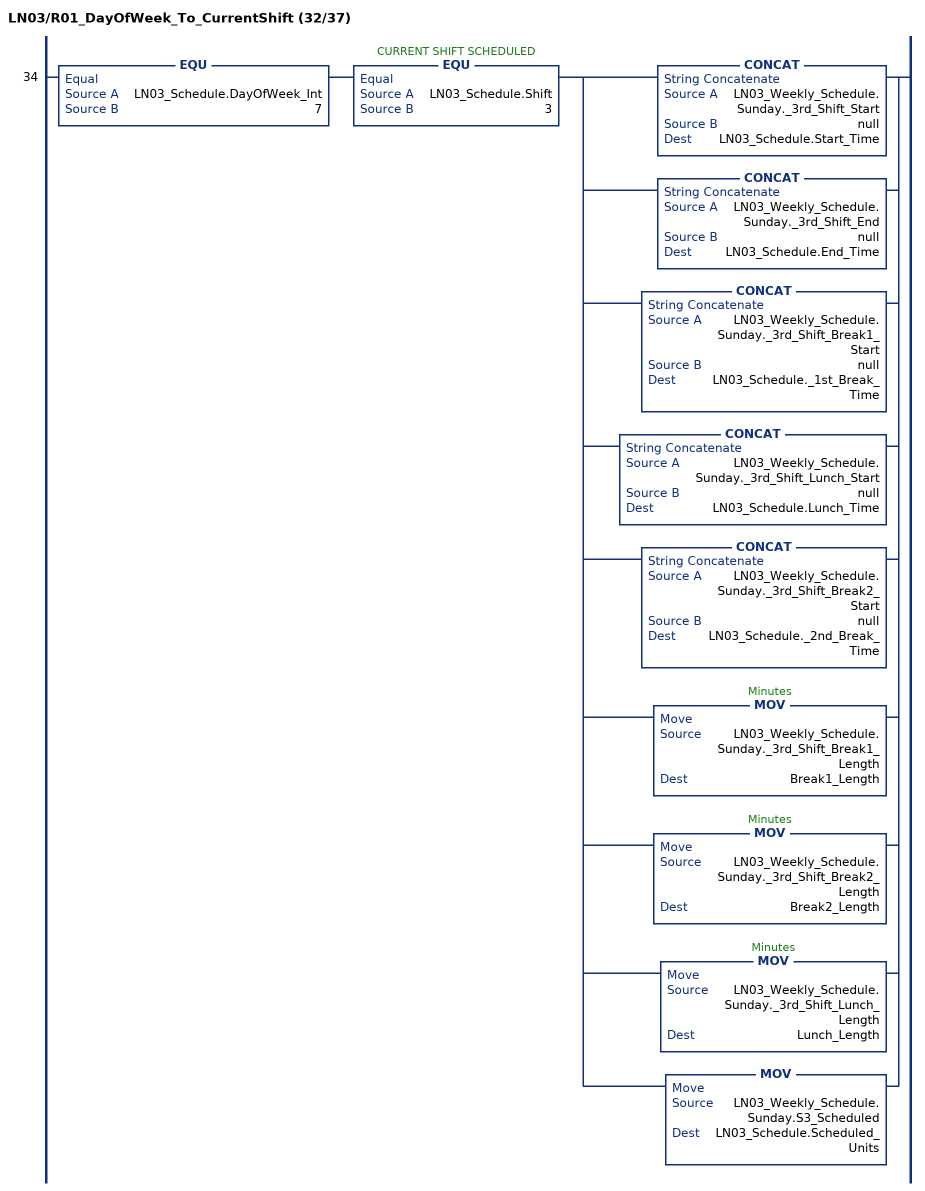
   34: EQU(LN03_Schedule.DayOfWeek_Int,7)EQU(LN03_Schedule.Shift,3)[CONCAT(LN03_Weekly_Schedule.Sunday._3rd_Shift_Start,null,LN03_Schedule.Start_Time) ,CONCAT(LN03_Weekly_Schedule.Sunday._3rd_Shift_End,null,LN03_Schedule.End_Time) ,CONCAT(LN03_Weekly_Schedule.Sunday._3rd_Shift_Break1_Start,null,LN03_Schedule._1st_Break_Time) ,CONCAT(LN03_Weekly_Schedule.Sunday._3rd_Shift_Lunch_Start,null,LN03_Schedule.Lunch_Time) ,CONCAT(LN03_Weekly_Schedule.Sunday._3rd_Shift_Break2_Start,null,LN03_Schedule._2nd_Break_Time) ,MOV(LN03_Weekly_Schedule.Sunday._3rd_Shift_Break1_Length,Break1_Length) ,MOV(LN03_Weekly_Schedule.Sunday._3rd_Shift_Break2_Length,Break2_Length) ,MOV(LN03_Weekly_Schedule.Sunday._3rd_Shift_Lunch_Length,Lunch_Length) ,MOV(LN03_Weekly_Schedule.Sunday.S3_Scheduled,LN03_Schedule.Scheduled_Units) ];
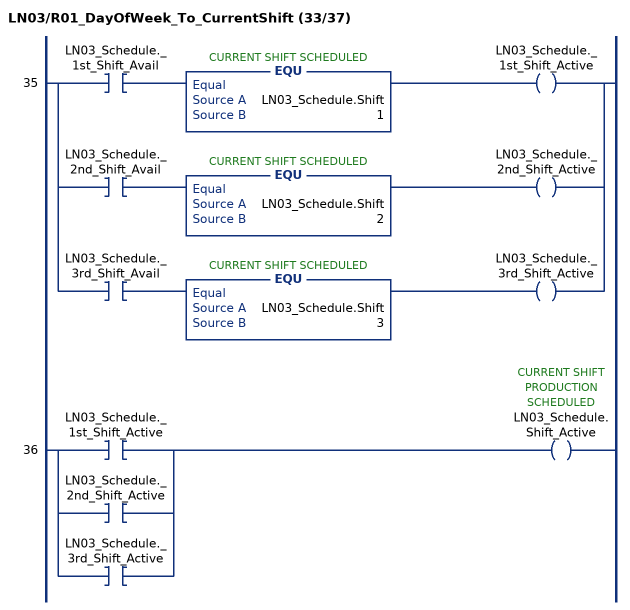
   35: [XIC(LN03_Schedule._1st_Shift_Avail) EQU(LN03_Schedule.Shift,1) OTE(LN03_Schedule._1st_Shift_Active) ,XIC(LN03_Schedule._2nd_Shift_Avail) EQU(LN03_Schedule.Shift,2) OTE(LN03_Schedule._2nd_Shift_Active) ,XIC(LN03_Schedule._3rd_Shift_Avail) EQU(LN03_Schedule.Shift,3) OTE(LN03_Schedule._3rd_Shift_Active) ];
   36: [XIC(LN03_Schedule._1st_Shift_Active) ,XIC(LN03_Schedule._2nd_Shift_Active) ,XIC(LN03_Schedule._3rd_Shift_Active) ]OTE(LN03_Schedule.Shift_Active);
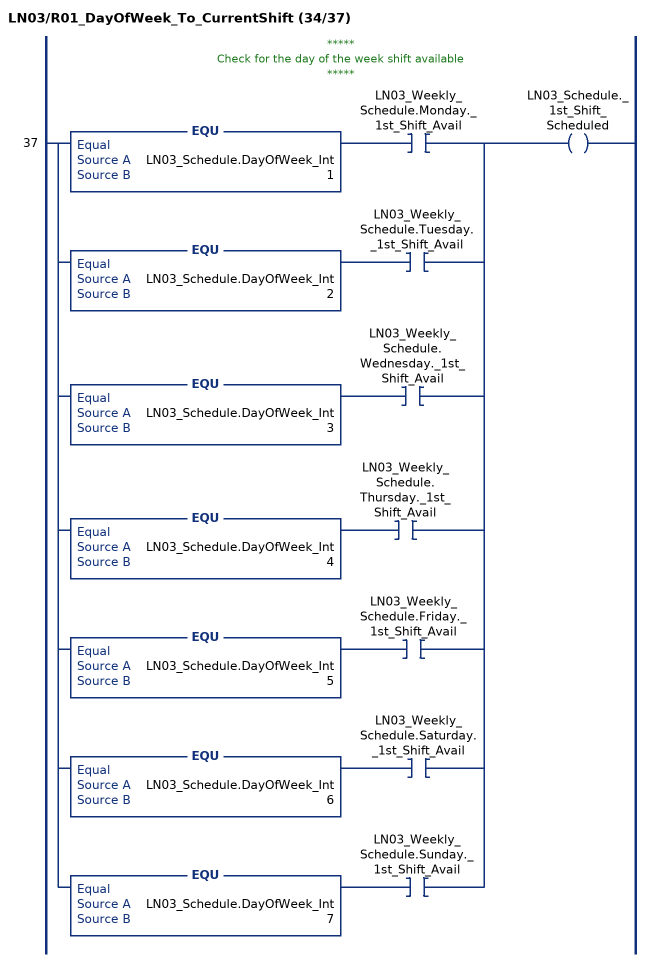
   // *****
   // Check for the day of the week shift available
   // *****
   37: [EQU(LN03_Schedule.DayOfWeek_Int,1) XIC(LN03_Weekly_Schedule.Monday._1st_Shift_Avail) ,EQU(LN03_Schedule.DayOfWeek_Int,2) XIC(LN03_Weekly_Schedule.Tuesday._1st_Shift_Avail) ,EQU(LN03_Schedule.DayOfWeek_Int,3) XIC(LN03_Weekly_Schedule.Wednesday._1st_Shift_Avail) ,EQU(LN03_Schedule.DayOfWeek_Int,4) XIC(LN03_Weekly_Schedule.Thursday._1st_Shift_Avail) ,EQU(LN03_Schedule.DayOfWeek_Int,5) XIC(LN03_Weekly_Schedule.Friday._1st_Shift_Avail) ,EQU(LN03_Schedule.DayOfWeek_Int,6) XIC(LN03_Weekly_Schedule.Saturday._1st_Shift_Avail) ,EQU(LN03_Schedule.DayOfWeek_Int,7) XIC(LN03_Weekly_Schedule.Sunday._1st_Shift_Avail) ]OTE(LN03_Schedule._1st_Shift_Scheduled);
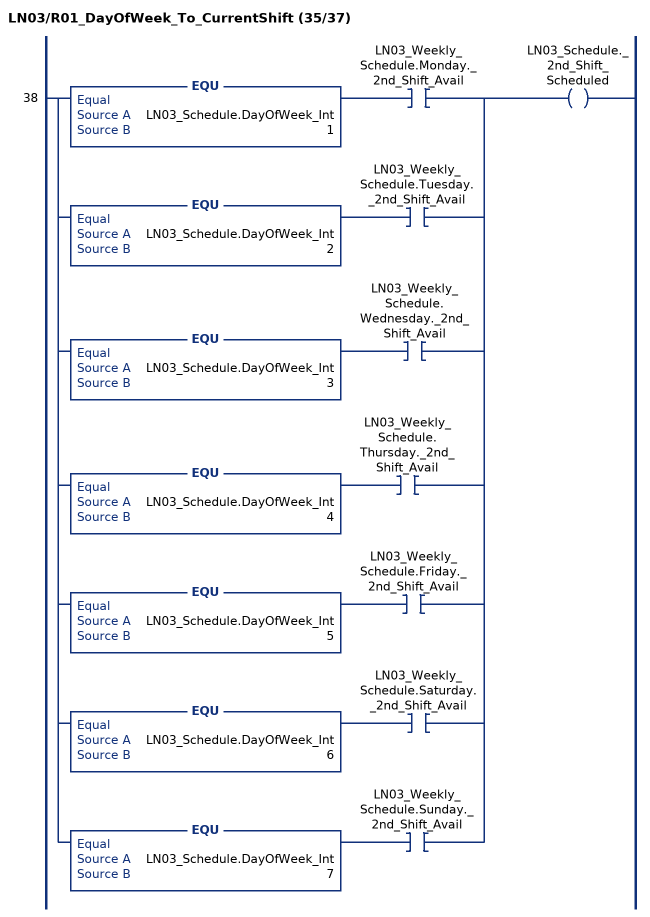
   38: [EQU(LN03_Schedule.DayOfWeek_Int,1) XIC(LN03_Weekly_Schedule.Monday._2nd_Shift_Avail) ,EQU(LN03_Schedule.DayOfWeek_Int,2) XIC(LN03_Weekly_Schedule.Tuesday._2nd_Shift_Avail) ,EQU(LN03_Schedule.DayOfWeek_Int,3) XIC(LN03_Weekly_Schedule.Wednesday._2nd_Shift_Avail) ,EQU(LN03_Schedule.DayOfWeek_Int,4) XIC(LN03_Weekly_Schedule.Thursday._2nd_Shift_Avail) ,EQU(LN03_Schedule.DayOfWeek_Int,5) XIC(LN03_Weekly_Schedule.Friday._2nd_Shift_Avail) ,EQU(LN03_Schedule.DayOfWeek_Int,6) XIC(LN03_Weekly_Schedule.Saturday._2nd_Shift_Avail) ,EQU(LN03_Schedule.DayOfWeek_Int,7) XIC(LN03_Weekly_Schedule.Sunday._2nd_Shift_Avail) ]OTE(LN03_Schedule._2nd_Shift_Scheduled);
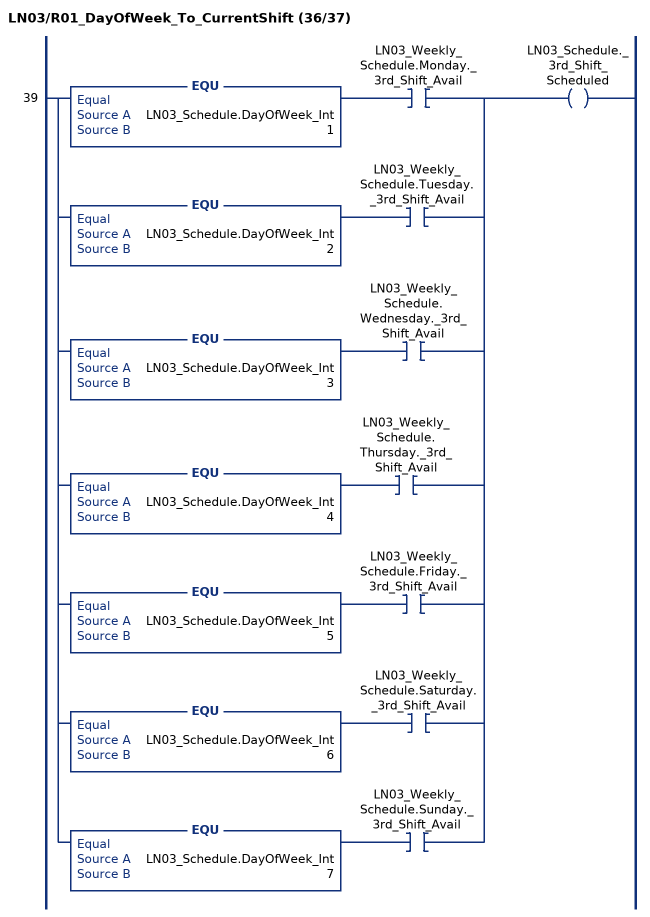
   39: [EQU(LN03_Schedule.DayOfWeek_Int,1) XIC(LN03_Weekly_Schedule.Monday._3rd_Shift_Avail) ,EQU(LN03_Schedule.DayOfWeek_Int,2) XIC(LN03_Weekly_Schedule.Tuesday._3rd_Shift_Avail) ,EQU(LN03_Schedule.DayOfWeek_Int,3) XIC(LN03_Weekly_Schedule.Wednesday._3rd_Shift_Avail) ,EQU(LN03_Schedule.DayOfWeek_Int,4) XIC(LN03_Weekly_Schedule.Thursday._3rd_Shift_Avail) ,EQU(LN03_Schedule.DayOfWeek_Int,5) XIC(LN03_Weekly_Schedule.Friday._3rd_Shift_Avail) ,EQU(LN03_Schedule.DayOfWeek_Int,6) XIC(LN03_Weekly_Schedule.Saturday._3rd_Shift_Avail) ,EQU(LN03_Schedule.DayOfWeek_Int,7) XIC(LN03_Weekly_Schedule.Sunday._3rd_Shift_Avail) ]OTE(LN03_Schedule._3rd_Shift_Scheduled);
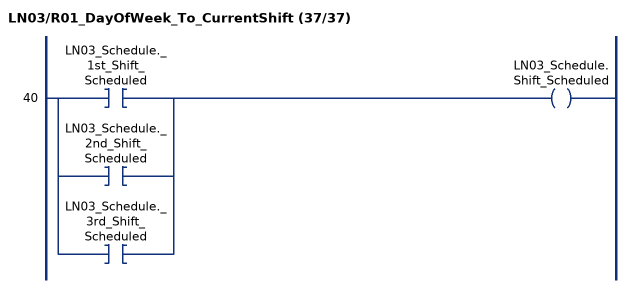
   40: [XIC(LN03_Schedule._1st_Shift_Scheduled) ,XIC(LN03_Schedule._2nd_Shift_Scheduled) ,XIC(LN03_Schedule._3rd_Shift_Scheduled) ]OTE(LN03_Schedule.Shift_Scheduled);
END_ROUTINE
